# EPICS substitutions: mc09/tpmacApp/pmc/xf16idc-mc09-brake.substitutions
file "PLC_brake.pmc"
{
pattern
{ PLC, BRAKE, MOTOR, APPLY, RELEASE }
{16,	32,	5,	0, 	1}
{17,    33,     8,	0,	1}
}
